{attribute 'qualified_only'}
{attribute 'strict'}
TYPE E_Severity :
(
	Error := 0,
	Warning := 1,
	Event := 2
);
END_TYPE

(* stored: Version 1.1.0.1
   DUT E_Severity: Id {40552126-6936-4685-b5e5-23ff426a1d04} *)
